// TIA Portal V19 export
TYPE "PositioningMachine_Par"
// stored: Access Published
   STRUCT
      PosTolerance : LReal;
      DelayInPosition : Time;
      Man : Struct
         VelBwd : LReal;
         VelFwdHigh : LReal;
         VelFwdLow : LReal;
         Acc : LReal;
         Dec : LReal;
         Jerk : LReal;
         DelayChangeVel : Time;
         UsePositionControl : Bool;
      END_STRUCT;
   END_STRUCT;
END_TYPE
